Staubli VAL3: camera.dtx

public num nErrorCode
public string sErrorMsg[121]
  [0] = "Login> Unrecognized command"
  [1] = "Login> Wrong user name or password"
  [2] = "Login> Communication Error"
  [10] = "Set Online> Command successfully"
  [11] = "Set Online> Unrecognized command"
  [12] = "Set Online> The value given for Int is either out of range, or is not a valid integer"
  [13] = "Set Online> The command could not be executed"
  [14] = "Set Online> Sensor is set Offline manually "
  [15] = "Set Online> User does not have Full Access to execute the command."
  [20] = "Get Online> The In-Sight sensor is currently Offline"
  [21] = "Get Online> The In-Sight sensor is currently Online"
  [30] = "Load File> Command successfully"
  [31] = "Load File> Unrecognized command"
  [32] = "Load File> The filename is missing"
  [33] = "Load File> The job failed to load, the sensor is Online, or the file was not found"
  [34] = "Load File> The job to be loaded was not found, or the sensor is out of memory"
  [35] = "Load File> User does not have Full Access"
  [40] = "get File> Command successfully"
  [41] = "get File> Unrecognized command"
  [42] = "get File> The active job has not been saved"
  [50] = "Save file> Command successfully"
  [51] = "Save file> Unrecognized command"
  [52] = "Save file> The filename is missing"
  [53] = "Save file>The job failed to save, the sensor is Online or the file was not found"
  [54] = "Save file> User does not have Full Access "
  [60] = "Set Event> Command successfully"
  [61] = "Set Event> Unrecognized command"
  [62] = "Set Event> The number is either out of range or not an integer"
  [63] = "Set Event>The command could not be executed, or the sensor is Offline"
  [64] = "Set Event> User does not have Full Access "
  [70] = "Get Value> Command successfully"
  [71] = "Get Value> Unrecognized command"
  [72] = "Get Value> Cell ID is invalid"
  [73] = "Get Value> The command could not be executed"
  [80] = "Set Float> Command successfully"
  [81] = "Set Float> Unrecognized command"
  [82] = "Set Float> Cell ID is invalid, or not a float"
  [83] = "Set Float> Cell was not created by the EditFloat function"
  [84] = "Set Float> User does not have Full Access "
  [90] = "Set Integer> Command successfully"
  [91] = "Set Integer>Unrecognized command"
  [92] = "Set Integer>Cell ID invalid, or not an integer"
  [93] = "Set Integer> Integer value is outside of the control's valid range or cell was not created by the EditInt function"
  [94] = "Set Integer> User does not have Full Access"
  [100] = "Set String> Command successfully"
  [101] = "Set String> Unrecognized command"
  [102] = "Set String> Cell ID invalid"
  [103] = "Set String> String is too longer or the cell does not contain an EditString function"
  [104] = "Set String> User does not have Full Access"
  [110] = "Cell Format> OK"
  [111] = "Cell Format> Invalid column"
  [112] = "Cell Format> Invalid row"
  [113] = "Cell Format> Row number out of range"
public sio sSocket
public bool bConnected
